FUNCTION DWORD_TO_WORDS
  (* Standard: 61499-1 *)
  (* Version 1.0, 2024-02-22, franz *)
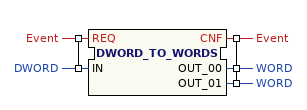
  EVENT_INPUT
    REQ WITH IN; (* Normal Execution Request *)
  END_EVENT
  EVENT_OUTPUT
    CNF WITH OUT_00, OUT_01; (* Execution Confirmation *)
  END_EVENT
  VAR_INPUT
    IN : DWORD; (* DWORD Input *)
  END_VAR
  VAR_OUTPUT
    OUT_00 : WORD; (* WORD 00 *)
    OUT_01 : WORD; (* WORD 01 *)
  END_VAR
  BODY IN ST:
FUNCTION DWORD_TO_WORDS

VAR_INPUT
	IN : DWORD;    // DWORD Input
END_VAR

VAR_OUTPUT
	OUT_00 : WORD;    // WORD 00
	OUT_01 : WORD;    // WORD 01
END_VAR

(* this Function extracts the 2 WORD from a dword *)
OUT_00 := DWORD_TO_WORD(SHR(IN AND DWORD_WORD_00, SHIFT_WORD_00));
OUT_01 := DWORD_TO_WORD(SHR(IN AND DWORD_WORD_01, SHIFT_WORD_01));

END_FUNCTION
  END_BODY
END_FUNCTION
